{attribute 'GeneratedUsingTerminal: EL3004-0000-0016'}
{attribute addProperty BoxType "EL3004-0000-0016"}
{attribute addProperty Id "AI_Standard_Channel_1AT %I*AI_Standard_Channel_EA9DF21E9AI_Standard_Channel_2AT %I*AI_Standard_Channel_EA9DF21E9AI_Standard_Channel_3AT %I*AI_Standard_Channel_EA9DF21E9AI_Standard_Channel_4AT %I*AI_Standard_Channel_EA9DF21E9WcStateAT %I*WcState_9091E0EB2InfoDataAT %I*InfoData_32EB74EA10"}
{attribute addProperty CRC "3893664799"}
{attribute addProperty Size "48"}
TYPE EL3004_E8149C1F EXTENDS EtcSlaveTerminalBase_947E5A46 :
STRUCT
	{attribute addProperty Name "AI_Standard_Channel_1"}
	AI_Standard_Channel_1 : AI_Standard_Channel_EA9DF21E;
	{attribute addProperty Name "AI_Standard_Channel_2"}
	AI_Standard_Channel_2 : AI_Standard_Channel_EA9DF21E;
	{attribute addProperty Name "AI_Standard_Channel_3"}
	AI_Standard_Channel_3 : AI_Standard_Channel_EA9DF21E;
	{attribute addProperty Name "AI_Standard_Channel_4"}
	AI_Standard_Channel_4 : AI_Standard_Channel_EA9DF21E;
	{attribute addProperty Name "WcState"}
	WcState : WcState_9091E0EB;
	{attribute addProperty Name "InfoData"}
	InfoData : InfoData_32EB74EA;
END_STRUCT
END_TYPE

(* stored: Version 1.2.0.0, ProductVersion 3.1.4024.9
   DUT EL3004_E8149C1F: Id {57ea50e2-1fa4-4039-81d2-ca0482ec9e84} *)
